(* CoDeSys 2.3.9.37 project: Cap6_6.pro *)
(* Libraries: Standard.lib 4.10.05 12:14:46 *)

(* POU PLC_PRG, LD *)
PROGRAM PLC_PRG
VAR
      (* Entradas *)
	Selec: BOOL;
	A: BOOL;
	B: BOOL;
       (* Salidas *)
	Luz: BOOL;
END_VAR
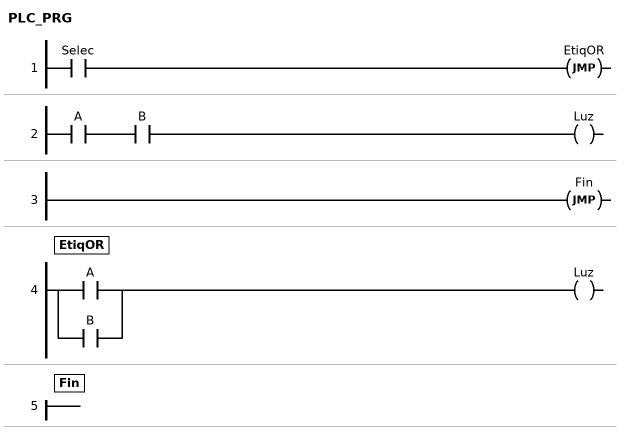
_LD_ (* Ladder Diagram *)
NETWORK 1
	[Selec] --- >>EtiqOR
NETWORK 2
	[A] - [B] --- (Luz)
NETWORK 3
	* --- >>Fin
NETWORK 4 EtiqOR:
	{ [A] | [B] } --- (Luz)
NETWORK 5 Fin:
	*
_END_LD_
(* the same logic as Structured Text *)
(* Network 1 *)
IF Selec THEN JMP EtiqOR; END_IF;
(* Network 2 *)
Luz := A AND B;
(* Network 3 *)
JMP Fin;
(* Network 4 *)
EtiqOR:
Luz := A OR B;
(* Network 5 *)
Fin:
END_PROGRAM

(* Visualisation Visu
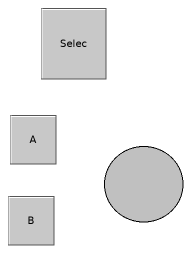
button at (81,23)-(146,94): text "Selec"; toggles PLC_PRG.Selec
button at (50,130)-(96,179): text "A"; toggles PLC_PRG.A
button at (48,211)-(94,260): text "B"; toggles PLC_PRG.B
ellipse at (144,161)-(223,237): alarm colour if PLC_PRG.Luz
*)
